TYPE palletParamsU :
STRUCT
	
	zeroPos             : REAL;
    moveDownStep		: REAL;
	moveUpStep 			: REAL;



END_STRUCT
END_TYPE

(* stored: Version 1.1.0.1, ProductVersion 3.1.4024.3
   DUT palletParamsU: Id {1ee5c8fc-3b85-4051-ab38-f95a42e3dd60} *)
